FUNCTION_BLOCK fbManipulatorContext  EXTENDS TcoCore.TcoContext
VAR
	_automat : fbManipulatorAutomat(THIS^, true); 
END_VAR

METHOD PROTECTED  Main
_automat();
END_METHOD

END_FUNCTION_BLOCK

(* stored: Version 1.1.0.1, ProductVersion 3.1.4024.6
   POU fbManipulatorContext: Id {fea94ac3-4856-422d-b18c-1c08797d1ff1}, SpecialFunc None
   Method Main: Id {cf5d8b8e-71ea-4109-8bb9-cf892a386f2d} *)
